SUBAPPLICATION Uebung_013 (* SR-Flip-Flop (Softkey) *)
  (* Standard: 61499-2 *)
  (* Version 1.0, 2023-10-23, franz *)
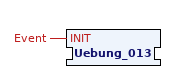
  EVENT_INPUT
    INIT;
  END_EVENT
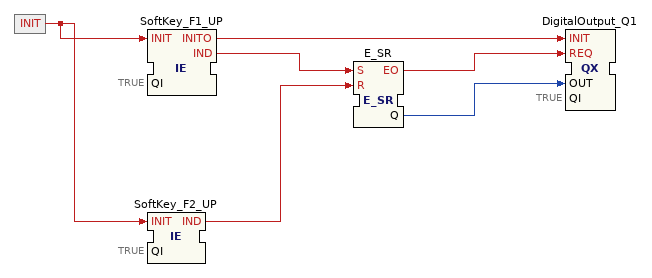
  FBS
    DigitalOutput_Q1 : QX(QI := TRUE);
    SoftKey_F1_UP : IE(QI := TRUE);
    SoftKey_F2_UP : IE(QI := TRUE);
    E_SR : E_SR;
  END_FBS
  EVENT_CONNECTIONS
    INIT TO SoftKey_F1_UP.INIT;
    SoftKey_F1_UP.INITO TO DigitalOutput_Q1.INIT;
    INIT TO SoftKey_F2_UP.INIT;
    SoftKey_F1_UP.IND TO E_SR.S;
    SoftKey_F2_UP.IND TO E_SR.R;
    E_SR.EO TO DigitalOutput_Q1.REQ;
  END_CONNECTIONS
  DATA_CONNECTIONS
    E_SR.Q TO DigitalOutput_Q1.OUT;
  END_CONNECTIONS
END_SUBAPPLICATION
